PROGRAM MAIN
VAR
	fbReadRegs	:	FB_MBReadRegs;
	bRead		:	BOOL;
	nValue		:	ARRAY[0..3] OF INT;
	M0	AT%MB0	:	ARRAY[0..3] OF WORD;

END_VAR

fbReadRegs(
	sIPAddr:='' , 
	nTCPPort:=502 , 
	nUnitID:=255 , 
	nQuantity:=4 , 
	nMBAddr:=16#3000 , 
	cbLength:= SIZEOF(nValue), 
	pDestAddr:= ADR(nValue) , 
	bExecute:=bRead, 
	tTimeout:=T#5S , 
	bBusy=> , 
	bError=> , 
	nErrId=> , 
	cbRead=> );

END_PROGRAM

(* stored: Version 1.1.0.1, ProductVersion 3.1.4022.18
   POU MAIN: Id {12f1c17e-484a-4f47-859b-178b01c50a7e}, SpecialFunc None *)
